(* PLC project PID, Beckhoff Automation GmbH TwinCAT PLC Control 3.5.13.21 *)
(* stored: creationDateTime 2022-05-16T15:08:28.8825399, modificationDateTime 2022-05-16T15:08:28.8825399 *)

FUNCTION_BLOCK FB_PT1T2_Process
VAR_INPUT
	u		: REAL;				// Aktuelle Steuergroesse
	Mode	: E_System_Mode;	// Aktueller Modus
	Param	: S_PT1T2_Param;	// Parameter vom PT1T2 Modell
	T		: REAL;				// Abtastzeit
END_VAR
VAR_OUTPUT
	y 		: REAL;				// Ausgangsgroesse
END_VAR
VAR
	a1		: REAL;
	a2		: REAL;
	b0 		: REAL;
	b1		: REAL;
	c1		: REAL;
	c2		: REAL;
	y_k_1	: REAL;
	y_k_2	: REAL;
	u_k_1	: REAL;
	u_k_2	: REAL;
END_VAR

            CASE Mode OF
	E_System_Mode.System_Init:
		// calculate coefficients
		a1 := EXP(-T/Param.T1);
		a2 := EXP(-T/Param.T2);
		b0 := (Param.K/(Param.T1-Param.T2))*(Param.T1*(1-a1)-Param.T2*(1-a2));
		b1 := (Param.K/(Param.T1-Param.T2))*(Param.T2*a1*(1-a2)-Param.T1*a2*(1-a1));;
		c1 := -(a1 + a2);
		c2 := a1 * a2;
		
	E_System_Mode.System_Run:
		// implements differencial equation
		y := b0*u_k_1 + b1*u_k_2 - c1*y_k_1 - c2*y_k_2;
		
		// store vars
		u_k_2 := u_k_1;
		u_k_1 := u;
		y_k_2 := y_k_1;
		y_k_1 := y;
		
	ELSE  // default assignment
	;
		
END_CASE
          
END_FUNCTION_BLOCK
